FUNCTION_BLOCK MyRender (* Function block to display and animate an Image *)
  (* Standard: 61499-2 *)
  (* Version 0.2, 2006-01-05, Anirudha, UoA, Added Layer attribute *)
  (* Version 0.1, 2005-12-04, Anirudha, UoA, Added Angle attribute *)
  (* Compiler header: package fb.rt.cs725; *)
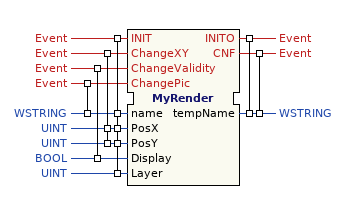
  EVENT_INPUT
    INIT WITH name, PosX, PosY, Layer; (* Initialization Request *)
    ChangeXY WITH PosX, PosY; (* Normal Execution Request *)
    ChangeValidity WITH Display;
    ChangePic WITH name;
  END_EVENT
  EVENT_OUTPUT
    INITO WITH tempName; (* Initialization Confirm *)
    CNF WITH tempName; (* Execution Confirmation *)
  END_EVENT
  VAR_INPUT
    name : WSTRING;
    PosX : UINT;
    PosY : UINT;
    Display : BOOL;
    Layer : UINT;
  END_VAR
  VAR_OUTPUT
    tempName : WSTRING;
  END_VAR
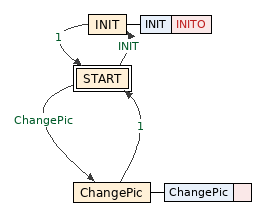
  EC_STATES
    START; (* Initial State *)
    INIT : INIT -> INITO; (* Initialization *)
    ChangePic : ChangePic;
  END_STATES
  EC_TRANSITIONS
    START TO INIT := INIT;
    INIT TO START := 1;
    START TO ChangePic := ChangePic;
    ChangePic TO START := 1;
  END_TRANSITIONS
  ALGORITHM INIT IN Java: (* Initialization algorithm *)
tempName.value = "/fb/rt/cs405/SSG.png";
System.out.println("My Render Init");
  END_ALGORITHM
  ALGORITHM ChangeXY IN ST:

  END_ALGORITHM
  ALGORITHM ChangeValidity IN ST:

  END_ALGORITHM
  ALGORITHM ChangePic IN Java:
if(!tempName.value.equals(name.value))
{
      //System.out.println("My Out Render ChangePic = " + name + "    " + tempName);
      tempName.value = name.value;
     // System.out.println("My Render ChangePic = " + name + "    " + tempName);
      CNF.serviceEvent(this);
}
//System.out.println("My Out1234567 Render ChangePic = " + name + "    " + tempName);
  END_ALGORITHM
END_FUNCTION_BLOCK
